// TIA Portal project "Simon_VTS_v0.2" (V15)

(* hardware
DEVICE "S71500/ET200MP station_1"  S7-1500 station
   slot 0: "Rail_0"  Rack  6ES7 590-1***0-0AA0
   slot 1: "PLC_1"  CPU 1511C-1 PN  6ES7 511-1CK00-0AB0  V2.1
      slot 3: "CPU display_1"  6ES7591-1AA00-0AA0
*)

// ===== PLC "PLC_1"  CPU 1511C-1 PN =====

VAR_GLOBAL   // PLC tag table "Default tag table"
   "System_Byte" AT %MB1 : Byte;
   "FirstScan" AT %M1.0 : Bool;
   "DiagStatusUpdate" AT %M1.1 : Bool;
   "AlwaysTRUE" AT %M1.2 : Bool;
   "AlwaysFALSE" AT %M1.3 : Bool;
   "Clock_Byte" AT %MB0 : Byte;
   "Clock_10Hz" AT %M0.0 : Bool;
   "Clock_5Hz" AT %M0.1 : Bool;
   "Clock_2.5Hz" AT %M0.2 : Bool;
   "Clock_2Hz" AT %M0.3 : Bool;
   "Clock_1.25Hz" AT %M0.4 : Bool;
   "Clock_1Hz" AT %M0.5 : Bool;
   "Clock_0.625Hz" AT %M0.6 : Bool;
   "Clock_0.5Hz" AT %M0.7 : Bool;
END_VAR

VAR_GLOBAL   // PLC tag table "IO"
   "ConveyorInPositionBit0" AT %I10.0 : Bool;
   "ConveyorInPositionBit1" AT %I10.1 : Bool;
   "ConveyorInPositionBit2" AT %I10.2 : Bool;
   "ConveyorInPositionBit3" AT %I10.3 : Bool;
   "RobotInPositionBit0" AT %I10.4 : Bool;
   "RobotInPositionBit1" AT %I10.5 : Bool;
   "RobotInPositionBit2" AT %I10.6 : Bool;
   "VakumOK" AT %I10.7 : Bool;
   "ProductIDBit0" AT %I11.0 : Bool;
   "ProductIDBit1" AT %I11.1 : Bool;
   "ProductIDBit2" AT %I11.2 : Bool;
   "ProductIDBit3" AT %I11.3 : Bool;
   "InicializationButton" AT %I11.4 : Bool;
   "StartButton" AT %I11.5 : Bool;
   "OrderBit0" AT %I11.6 : Bool;
   "OrderBit1" AT %I11.7 : Bool;
   "ConveyorMoveBit0" AT %Q4.0 : Bool;
   "ConveyorMoveBit1" AT %Q4.1 : Bool;
   "ConveyorMoveBit2" AT %Q4.2 : Bool;
   "ConveyorMoveBit3" AT %Q4.3 : Bool;
   "ConveyorStart" AT %Q4.4 : Bool;
   "RobotMoveBit0" AT %Q4.5 : Bool;
   "RobotMoveBit1" AT %Q4.6 : Bool;
   "RobotMoveBit2" AT %Q4.7 : Bool;
   "RobotStart" AT %Q5.0 : Bool;
   "VacuumStart" AT %Q5.1 : Bool;
   "CameraTrigger" AT %Q5.2 : Bool;
   "SingnalTowerBlue" AT %Q5.3 : Bool;
   "SingnalTowerYellow" AT %Q5.4 : Bool;
END_VAR

DATA_BLOCK "DB_TEST"   // DB1
{ S7_Optimized_Access := 'TRUE' }
VERSION : 0.1
   VAR
      bOrderBit0 : Bool := TRUE;
      bOrderBit1 : Bool;
   END_VAR
BEGIN
END_DATA_BLOCK

DATA_BLOCK "DB_MainControl"   // DB100
{ S7_Optimized_Access := 'TRUE' }
VERSION : 0.1
// stored: InstanceOfName FB_MainControl
"FB_MainControl"
BEGIN
END_DATA_BLOCK

FUNCTION_BLOCK "FB_MainControl"   // FB100, SCL
{ S7_Optimized_Access := 'TRUE' }
VERSION : 0.1
   VAR_INPUT
      bConveyorInPositionBit0 : Bool;
      bConveyorInPositionBit1 : Bool;
      bConveyorInPositionBit2 : Bool;
      bConveyorInPositionBit3 : Bool;
      bRobotInPositionBit0 : Bool;
      bRobotInPositionBit1 : Bool;
      bRobotInPositionBit2 : Bool;
      bVacuumOK : Bool;
      bProductIDBit0 : Bool;
      bProductIDBit1 : Bool;
      bProductIDBit2 : Bool;
      bProductIDBit3 : Bool;
      bInicializationButton : Bool;
      bStartButton : Bool;
      bOrderBit0 : Bool;
      bOrderBit1 : Bool;
   END_VAR
   VAR_OUTPUT
      bConveyorMoveBit0 : Bool;
      bConveyorMoveBit1 : Bool;
      bConveyorMoveBit2 : Bool;
      bConveyorMoveBit3 : Bool;
      bConveyorStart : Bool;
      bRobotMoveBit0 : Bool;
      bRobotMoveBit1 : Bool;
      bRobotMoveBit2 : Bool;
      bRobotStart : Bool;
      bVacuumStart : Bool;
      bCameraTrigger : Bool;
      bSingnalTowerBlue : Bool;
      bSingnalTowerYellow : Bool;
      bInInicalPosition : Bool;
   END_VAR
   VAR
      BConveyorInPosition : Byte;
      iConveyorInPosition : Int;
      BRobotInPosition : Byte;
      iRobotInPosition : Int;
      BProduct : Byte;
      iProduct : Int;
      BConveyorMove : Byte;
      iConveyorMove : Int;
      BRobotMove : Byte;
      iRobotMove : Int;
      rtInicialization : R_TRIG;
      rtStart : R_TRIG;
      iFSM : Int;
      tonDelay_1 : TON_TIME;
      iPositionTemp : Int;
      iConveyorPositionTemp : Int;
      iBasket_1 : Int;
      iBasket_2 : Int;
      iBasket_3 : Int;
      iSignalTower : Int;
      arrConveyorPosition : Array[1..10] of Int;
      arrConveyorConntent : Array[1..10] of Int;
      arrEmpty : Array[1..10] of Int;
      arrRecipe : Array[0..3] of Int;
   END_VAR
   VAR_TEMP
      i : Int;
   END_VAR
   VAR CONSTANT
      tDelayTime_1 : Time := T#250ms;
   END_VAR
   // arrConveyorPosition[1] := 10;
   // arrConveyorPosition[2] := 1;
   // arrConveyorPosition[3] := 2;
   // arrConveyorPosition[4] := 3;
   // arrConveyorPosition[5] := 4;
   // arrConveyorPosition[6] := 5;
   // arrConveyorPosition[7] := 6;
   // arrConveyorPosition[8] := 7;
   // arrConveyorPosition[9] := 8;
   // arrConveyorPosition[10] := 9;
   // arrEmpty[1] := 0;
   // arrEmpty[2] := 0;
   // arrEmpty[3] := 0;
   // arrEmpty[4] := 0;
   // arrEmpty[5] := 0;
   // arrEmpty[6] := 0;
   // arrEmpty[7] := 0;
   // arrEmpty[8] := 0;
   // arrEmpty[9] := 0;
   // arrEmpty[10] := 0;
BEGIN
   #BConveyorInPosition.%X0 := #bConveyorInPositionBit0;
   #BConveyorInPosition.%X1 := #bConveyorInPositionBit1;
   #BConveyorInPosition.%X2 := #bConveyorInPositionBit2;
   #BConveyorInPosition.%X3 := #bConveyorInPositionBit3;
   #iConveyorInPosition := BYTE_TO_INT(#BConveyorInPosition);

   #BRobotInPosition.%X0 := #bRobotInPositionBit0;
   #BRobotInPosition.%X1 := #bRobotInPositionBit1;
   #BRobotInPosition.%X2 := #bRobotInPositionBit2;
   #iRobotInPosition := BYTE_TO_INT(#BRobotInPosition);

   #BProduct.%X0 := #bProductIDBit0;
   #BProduct.%X1 := #bProductIDBit1;
   #BProduct.%X2 := #bProductIDBit2;
   #BProduct.%X3 := #bProductIDBit3;
   #iProduct := BYTE_TO_INT(#BProduct);

   IF NOT #bOrderBit0 AND NOT #bOrderBit1 THEN
       #arrRecipe[0] := 0;
       #arrRecipe[1] := 0;
       #arrRecipe[2] := 0;
       #arrRecipe[3] := 0;
   ELSIF NOT #bOrderBit0 AND #bOrderBit1 THEN
       #arrRecipe[0] := 10;
       #arrRecipe[1] := 30;
       #arrRecipe[2] := 20;
       #arrRecipe[3] := 30;
   ELSIF #bOrderBit0 AND NOT #bOrderBit1 THEN
       #arrRecipe[0] := 30;
       #arrRecipe[1] := 20;
       #arrRecipe[2] := 10;
       #arrRecipe[3] := 30;
   ELSIF #bOrderBit0 AND #bOrderBit1 THEN
       #arrRecipe[0] := 10;
       #arrRecipe[1] := 20;
       #arrRecipe[2] := 30;
       #arrRecipe[3] := 30;
   END_IF;


   //Start initialization position movement.
   #rtInicialization(CLK:=#bInicializationButton);
   IF #rtInicialization.Q THEN
       #iFSM := 10;
       #bInInicalPosition := FALSE;
   END_IF;

   #rtStart(CLK := #bStartButton);
   //Start sorting task
   IF #bInInicalPosition AND #rtStart.Q THEN
       #iFSM := 40;
       #bInInicalPosition := FALSE;
   END_IF;


   CASE #iFSM OF
       0:
           #bConveyorStart := FALSE;
           #iConveyorMove := 0;
           #bRobotStart := FALSE;
           #iRobotMove := 0;
           #tonDelay_1(IN := FALSE,
                       PT := #tDelayTime_1);
           #arrConveyorConntent := #arrEmpty;
           #bVacuumStart := FALSE;
           #iBasket_1 := 0;
           ;
       10:
           #iFSM := 20;
           #bConveyorStart := FALSE;
           #iConveyorMove := 0;
           #bRobotStart := FALSE;
           #iRobotMove := 0;
           #tonDelay_1(IN := FALSE,
                       PT := #tDelayTime_1);
           #iSignalTower := 1;
           ;
       20:
           //Robot initial position movment
           IF #iRobotInPosition = 7 THEN
               #iFSM := 30;
               #bRobotStart := FALSE;
               #iRobotMove := 0;
               #tonDelay_1(IN := FALSE,
                           PT := #tDelayTime_1);
           ELSE
               #iRobotMove := 7;
               #tonDelay_1(IN := TRUE,
                           PT := #tDelayTime_1);
               #bRobotStart := #tonDelay_1.Q;
           END_IF;
           ;
       30:
           //Conveyor initial position movment
           IF #iConveyorInPosition = 15 THEN
               #iFSM := 0;
               #bInInicalPosition := TRUE;
               #bConveyorStart := FALSE;
               #iConveyorMove := 0;
               #tonDelay_1(IN := FALSE,
                           PT := #tDelayTime_1);
           ELSE
               #iConveyorMove := 15;
               #tonDelay_1(IN := TRUE,
                           PT := #tDelayTime_1);
               #bConveyorStart := #tonDelay_1.Q;
           END_IF;
           ;
       40:
           #iFSM := 50;
           #iPositionTemp := 1;
           #iSignalTower := 2;
           ;

       50:
           //Move to DMC read position.
           IF #iPositionTemp < 11 THEN
               #iConveyorMove := #arrConveyorPosition[#iPositionTemp];
               #tonDelay_1(IN := TRUE,
                           PT := #tDelayTime_1);
               #bConveyorStart := #tonDelay_1.Q;

               IF #iConveyorInPosition = #arrConveyorPosition[#iPositionTemp] THEN
                   #iFSM := 60;
                   #iConveyorMove := 0;
                   #tonDelay_1(IN := FALSE,
                               PT := #tDelayTime_1);
                   #bConveyorStart := FALSE;
               END_IF;
           ELSE
               #iFSM := 70;
               #iPositionTemp := 0;
           END_IF;
           ;
       60:
           //DMC read.
           #bCameraTrigger := TRUE;
           IF #iProduct <> 0 THEN
               IF #iProduct = 3 OR #iProduct = 6 OR #iProduct = 9 THEN
                   #arrConveyorConntent[#iPositionTemp] := 10;
               ELSIF #iProduct = 1 OR #iProduct = 4 OR #iProduct = 7 THEN
                   #arrConveyorConntent[#iPositionTemp] := 20;
               ELSIF #iProduct = 2 OR #iProduct = 5 OR #iProduct = 8 OR #iProduct = 10 THEN
                   #arrConveyorConntent[#iPositionTemp] := 30;
               ELSE
                   #arrConveyorConntent[#iPositionTemp] := 0;
               END_IF;
               #iPositionTemp := #iPositionTemp + 1;
               #bCameraTrigger := FALSE;
               #iFSM := 50;
           END_IF;
           ;
       70:
           //Robot home position movment
           IF #iRobotInPosition = 1 THEN
               #iFSM := 80;
               #bRobotStart := FALSE;
               #iRobotMove := 0;
               #tonDelay_1(IN := FALSE,
                           PT := #tDelayTime_1);
           ELSE
               #iRobotMove := 1;
               #tonDelay_1(IN := TRUE,
                           PT := #tDelayTime_1);
               #bRobotStart := #tonDelay_1.Q;
           END_IF;
           ;
       80:
           //Fist basket fill, fine part location.
           FOR #i := 1 TO 10 DO
               IF #iBasket_1 = 0 THEN
                   IF #arrConveyorConntent[#i] = 10 THEN
                       #iConveyorPositionTemp := #i;
                       #arrConveyorConntent[#i] := 0;
                       #iFSM := 90;
                       EXIT;
                   END_IF;
               ELSIF #iBasket_1 = 1 THEN
                   IF #arrConveyorConntent[#i] = 30 THEN
                       #iConveyorPositionTemp := #i;
                       #arrConveyorConntent[#i] := 0;
                       #iFSM := 90;
                       EXIT;
                   END_IF;
               ELSIF #iBasket_1 = 2 THEN
                   IF #arrConveyorConntent[#i] = 20 THEN
                       #iConveyorPositionTemp := #i;
                       #arrConveyorConntent[#i] := 0;
                       #iFSM := 90;
                       EXIT;
                   END_IF;
               END_IF;
           END_FOR;
           ;
       90:
           //Move conveyor to pickup position.
           IF #iConveyorInPosition = #iConveyorPositionTemp THEN
               #iFSM := 100;
               #iConveyorPositionTemp := 0;
               #bConveyorStart := FALSE;
               #iConveyorMove := 0;
               #tonDelay_1(IN := FALSE,
                           PT := #tDelayTime_1);
           ELSE
               #iConveyorMove := #iConveyorPositionTemp;
               #tonDelay_1(IN := TRUE,
                           PT := #tDelayTime_1);
               #bConveyorStart := #tonDelay_1.Q;
           END_IF;
           ;
       100:
           //Move to pickup position
           #bVacuumStart := TRUE;
           IF #iRobotInPosition = 2 THEN
               IF #bVacuumOK THEN
                   #iFSM := 110;
                   #bRobotStart := FALSE;
                   #iRobotMove := 0;
                   #tonDelay_1(IN := FALSE,
                               PT := #tDelayTime_1);
               END_IF;
           ELSE
               #iRobotMove := 2;
               #tonDelay_1(IN := TRUE,
                           PT := #tDelayTime_1);
               #bRobotStart := #tonDelay_1.Q;
           END_IF;
           ;
       110:
           //Move to basket 1
           IF #iRobotInPosition = 4 THEN
               IF #bVacuumOK THEN
                   #bRobotStart := FALSE;
                   #iRobotMove := 0;
                   #tonDelay_1(IN := FALSE,
                               PT := #tDelayTime_1);
                   #bVacuumStart := FALSE;
                   #iBasket_1 := #iBasket_1 + 1;
                   IF #iBasket_1 = 3 THEN
                       #iFSM := 130;
                   ELSE
                       #iFSM := 80;
                   END_IF;
               END_IF;
           ELSE
               #iRobotMove := 4;
               #tonDelay_1(IN := TRUE,
                           PT := #tDelayTime_1);
               #bRobotStart := #tonDelay_1.Q;
           END_IF;
           ;
       120:
           #arrConveyorConntent := #arrEmpty;
           #bRobotStart := FALSE;
           #iRobotMove := 0;
           #tonDelay_1(IN := FALSE,
                       PT := #tDelayTime_1);
           #bVacuumStart := FALSE;
           #iBasket_1 := 0;
           #iBasket_2 := 0;
           #iBasket_3 := 0;
           #iFSM := 0;
       130:
           //Second basket fill, fine part location.
           #iSignalTower := 3;
           FOR #i := 1 TO 10 DO
               IF #iBasket_2 = 0 THEN
                   IF #arrConveyorConntent[#i] = 20 THEN
                       #iConveyorPositionTemp := #i;
                       #arrConveyorConntent[#i] := 0;
                       #iFSM := 140;
                       EXIT;
                   END_IF;
               ELSIF #iBasket_2 = 1 THEN
                   IF #arrConveyorConntent[#i] = 10 THEN
                       #iConveyorPositionTemp := #i;
                       #arrConveyorConntent[#i] := 0;
                       #iFSM := 140;
                       EXIT;
                   END_IF;
               ELSIF #iBasket_2 = 2 THEN
                   IF #arrConveyorConntent[#i] = 30 THEN
                       #iConveyorPositionTemp := #i;
                       #arrConveyorConntent[#i] := 0;
                       #iFSM := 140;
                       EXIT;
                   END_IF;
               END_IF;
           END_FOR;
           ;
       140:
           //Move conveyor to pickup position.
           IF #iConveyorInPosition = #iConveyorPositionTemp THEN
               #iFSM := 150;
               #iConveyorPositionTemp := 0;
               #bConveyorStart := FALSE;
               #iConveyorMove := 0;
               #tonDelay_1(IN := FALSE,
                           PT := #tDelayTime_1);
           ELSE
               #iConveyorMove := #iConveyorPositionTemp;
               #tonDelay_1(IN := TRUE,
                           PT := #tDelayTime_1);
               #bConveyorStart := #tonDelay_1.Q;
           END_IF;
           ;
       150:
           //Move to pickup position
           #bVacuumStart := TRUE;
           IF #iRobotInPosition = 2 THEN
               IF #bVacuumOK THEN
                   #iFSM := 160;
                   #bRobotStart := FALSE;
                   #iRobotMove := 0;
                   #tonDelay_1(IN := FALSE,
                               PT := #tDelayTime_1);
               END_IF;
           ELSE
               #iRobotMove := 2;
               #tonDelay_1(IN := TRUE,
                           PT := #tDelayTime_1);
               #bRobotStart := #tonDelay_1.Q;
           END_IF;
           ;
       160:
           //Move to basket 2
           IF #iRobotInPosition = 5 THEN
               IF #bVacuumOK THEN
                   #bRobotStart := FALSE;
                   #iRobotMove := 0;
                   #tonDelay_1(IN := FALSE,
                               PT := #tDelayTime_1);
                   #bVacuumStart := FALSE;
                   #iBasket_2 := #iBasket_2 + 1;
                   IF #iBasket_2 = 3 THEN
                       #iFSM := 170;
                   ELSE
                       #iFSM := 130;
                   END_IF;
               END_IF;
           ELSE
               #iRobotMove := 5;
               #tonDelay_1(IN := TRUE,
                           PT := #tDelayTime_1);
               #bRobotStart := #tonDelay_1.Q;
           END_IF;
           ;
       170:
           //Thrd basket fill, fine part location.
           #iSignalTower := 4;
           FOR #i := 1 TO 10 DO
               IF #iBasket_3 = 0 THEN
                   IF #arrConveyorConntent[#i] = #arrRecipe[0] THEN
                       #iConveyorPositionTemp := #i;
                       #arrConveyorConntent[#i] := 0;
                       #iFSM := 180;
                       EXIT;
                   END_IF;
               ELSIF #iBasket_3 = 1 THEN
                   IF #arrConveyorConntent[#i] = #arrRecipe[1] THEN
                       #iConveyorPositionTemp := #i;
                       #arrConveyorConntent[#i] := 0;
                       #iFSM := 180;
                       EXIT;
                   END_IF;
               ELSIF #iBasket_3 = 2 THEN
                   IF #arrConveyorConntent[#i] = #arrRecipe[2] THEN
                       #iConveyorPositionTemp := #i;
                       #arrConveyorConntent[#i] := 0;
                       #iFSM := 180;
                       EXIT;
                   END_IF;
               ELSIF #iBasket_3 = 3 THEN
                   IF #arrConveyorConntent[#i] = #arrRecipe[3] THEN
                       #iConveyorPositionTemp := #i;
                       #arrConveyorConntent[#i] := 0;
                       #iFSM := 180;
                       EXIT;
                   END_IF;
               END_IF;
           END_FOR;
           ;
       180:
           //Move conveyor to pickup position.
           IF #iConveyorInPosition = #iConveyorPositionTemp THEN
               #iFSM := 190;
               #iConveyorPositionTemp := 0;
               #bConveyorStart := FALSE;
               #iConveyorMove := 0;
               #tonDelay_1(IN := FALSE,
                           PT := #tDelayTime_1);
           ELSE
               #iConveyorMove := #iConveyorPositionTemp;
               #tonDelay_1(IN := TRUE,
                           PT := #tDelayTime_1);
               #bConveyorStart := #tonDelay_1.Q;
           END_IF;
           ;
       190:
           //Move to pickup position
           #bVacuumStart := TRUE;
           IF #iRobotInPosition = 2 THEN
               IF #bVacuumOK THEN
                   #iFSM := 200;
                   #bRobotStart := FALSE;
                   #iRobotMove := 0;
                   #tonDelay_1(IN := FALSE,
                               PT := #tDelayTime_1);
               END_IF;
           ELSE
               #iRobotMove := 2;
               #tonDelay_1(IN := TRUE,
                           PT := #tDelayTime_1);
               #bRobotStart := #tonDelay_1.Q;
           END_IF;
           ;
           ;
       200:
           //Move to basket 3
           IF #iRobotInPosition = 6 THEN
               IF #bVacuumOK THEN
                   #bRobotStart := FALSE;
                   #iRobotMove := 0;
                   #tonDelay_1(IN := FALSE,
                               PT := #tDelayTime_1);
                   #bVacuumStart := FALSE;
                   #iBasket_3 := #iBasket_3 + 1;
                   IF #iBasket_3 = 4 THEN
                       #iFSM := 120;
                       #iSignalTower := 5;
                   ELSE
                       #iFSM := 170;
                   END_IF;
               END_IF;
           ELSE
               #iRobotMove := 6;
               #tonDelay_1(IN := TRUE,
                           PT := #tDelayTime_1);
               #bRobotStart := #tonDelay_1.Q;
           END_IF;
           ;
   END_CASE;


   IF #iSignalTower = 1 THEN
       #bSingnalTowerBlue := "Clock_0.5Hz";
       #bSingnalTowerYellow := "Clock_1Hz";
   ELSIF #iSignalTower = 2 OR #iSignalTower = 4 THEN
       #bSingnalTowerBlue := TRUE;
       #bSingnalTowerYellow := FALSE;
   ELSIF #iSignalTower = 3 THEN
       #bSingnalTowerBlue := FALSE;
       #bSingnalTowerYellow := "Clock_0.5Hz";
   ELSIF #iSignalTower = 5 THEN
       #bSingnalTowerBlue := "Clock_0.5Hz";
       #bSingnalTowerYellow := "Clock_0.5Hz";
   ELSE
       #bSingnalTowerBlue := FALSE;
       #bSingnalTowerYellow := FALSE;
   END_IF;








   #BConveyorMove := INT_TO_BYTE(#iConveyorMove);
   #bConveyorMoveBit0 := #BConveyorMove.%X0;
   #bConveyorMoveBit1 := #BConveyorMove.%X1;
   #bConveyorMoveBit2 := #BConveyorMove.%X2;
   #bConveyorMoveBit3 := #BConveyorMove.%X3;

   #BRobotMove := INT_TO_BYTE(#iRobotMove);
   #bRobotMoveBit0 := #BRobotMove.%X0;
   #bRobotMoveBit1 := #BRobotMove.%X1;
   #bRobotMoveBit2 := #BRobotMove.%X2;
END_FUNCTION_BLOCK

ORGANIZATION_BLOCK "Main"   // OB1, LAD, ProgramCycle
TITLE = "Main Program Sweep (Cycle)"
{ S7_Optimized_Access := 'TRUE' }
VERSION : 0.1
   VAR_INPUT
      Initial_Call : Bool;   // Initial call of this OB
      Remanence : Bool;   // =True, if remanent data are available
   END_VAR
BEGIN

REGION Network 1
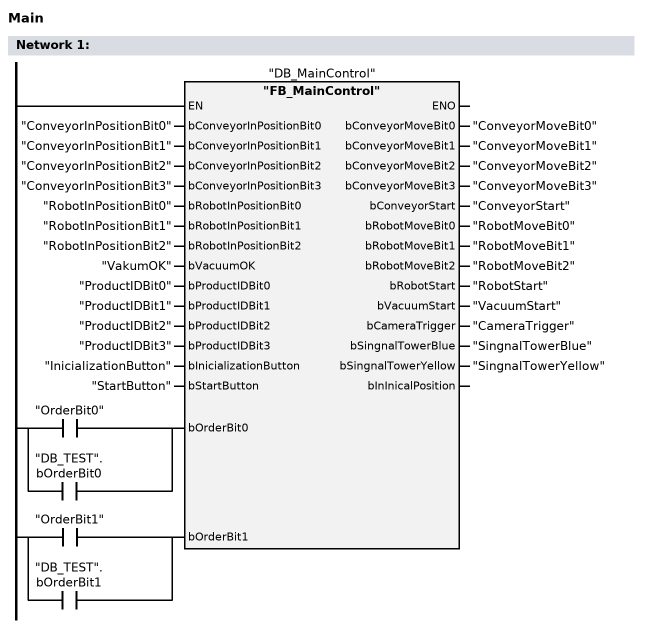
   RUNG wire#powerrail
      "DB_MainControl"(bOrderBit0 := wire#w1, bOrderBit1 := wire#w2, bConveyorInPositionBit0 := "ConveyorInPositionBit0", bConveyorInPositionBit1 := "ConveyorInPositionBit1", bConveyorInPositionBit2 := "ConveyorInPositionBit2", bConveyorInPositionBit3 := "ConveyorInPositionBit3", bRobotInPositionBit0 := "RobotInPositionBit0", bRobotInPositionBit1 := "RobotInPositionBit1", bRobotInPositionBit2 := "RobotInPositionBit2", bVacuumOK := "VakumOK", bProductIDBit0 := "ProductIDBit0", bProductIDBit1 := "ProductIDBit1", bProductIDBit2 := "ProductIDBit2", bProductIDBit3 := "ProductIDBit3", bInicializationButton := "InicializationButton", bStartButton := "StartButton", bConveyorMoveBit0 => "ConveyorMoveBit0", bConveyorMoveBit1 => "ConveyorMoveBit1", bConveyorMoveBit2 => "ConveyorMoveBit2", bConveyorMoveBit3 => "ConveyorMoveBit3", bConveyorStart => "ConveyorStart", bRobotMoveBit0 => "RobotMoveBit0", bRobotMoveBit1 => "RobotMoveBit1", bRobotMoveBit2 => "RobotMoveBit2", bRobotStart => "RobotStart", bVacuumStart => "VacuumStart", bCameraTrigger => "CameraTrigger", bSingnalTowerBlue => "SingnalTowerBlue", bSingnalTowerYellow => "SingnalTowerYellow", bInInicalPosition =>)
   END_RUNG
   RUNG wire#powerrail
      Contact( "OrderBit0" )
   END_RUNG wire#w1
   RUNG wire#powerrail
      Contact( "DB_TEST".bOrderBit0 )
   END_RUNG wire#w1
   RUNG wire#powerrail
      Contact( "OrderBit1" )
   END_RUNG wire#w2
   RUNG wire#powerrail
      Contact( "DB_TEST".bOrderBit1 )
   END_RUNG wire#w2
   // the same network as SCL:
   "DB_MainControl"(bConveyorInPositionBit0 := "ConveyorInPositionBit0",   // "FB_MainControl"
                    bConveyorInPositionBit1 := "ConveyorInPositionBit1",
                    bConveyorInPositionBit2 := "ConveyorInPositionBit2",
                    bConveyorInPositionBit3 := "ConveyorInPositionBit3",
                    bRobotInPositionBit0 := "RobotInPositionBit0",
                    bRobotInPositionBit1 := "RobotInPositionBit1",
                    bRobotInPositionBit2 := "RobotInPositionBit2",
                    bVacuumOK := "VakumOK",
                    bProductIDBit0 := "ProductIDBit0",
                    bProductIDBit1 := "ProductIDBit1",
                    bProductIDBit2 := "ProductIDBit2",
                    bProductIDBit3 := "ProductIDBit3",
                    bInicializationButton := "InicializationButton",
                    bStartButton := "StartButton",
                    bOrderBit0 := "OrderBit0" OR "DB_TEST".bOrderBit0,
                    bOrderBit1 := "OrderBit1" OR "DB_TEST".bOrderBit1,
                    bConveyorMoveBit0 => "ConveyorMoveBit0",
                    bConveyorMoveBit1 => "ConveyorMoveBit1",
                    bConveyorMoveBit2 => "ConveyorMoveBit2",
                    bConveyorMoveBit3 => "ConveyorMoveBit3",
                    bConveyorStart => "ConveyorStart",
                    bRobotMoveBit0 => "RobotMoveBit0",
                    bRobotMoveBit1 => "RobotMoveBit1",
                    bRobotMoveBit2 => "RobotMoveBit2",
                    bRobotStart => "RobotStart",
                    bVacuumStart => "VacuumStart",
                    bCameraTrigger => "CameraTrigger",
                    bSingnalTowerBlue => "SingnalTowerBlue",
                    bSingnalTowerYellow => "SingnalTowerYellow");
END_REGION
END_ORGANIZATION_BLOCK